KUKA KRL program: HmiToolCheck.src

&ACCESS RVP
&REL 18
&PARAM EDITMASK = *
&PARAM TEMPLATE = C:\KRC\Roboter\Template\vorgabe
DEF HmiToolCheck( )
;FOLD INI;%{PE}
  ;FOLD BASISTECH INI
    GLOBAL INTERRUPT DECL 3 WHEN $STOPMESS==TRUE DO IR_STOPM ( )
    INTERRUPT ON 3
    BAS (#INITMOV,0 )
  ;ENDFOLD (BASISTECH INI)
  ;FOLD USER INI
    ;Make your modifications here

  ;ENDFOLD (USER INI)
;ENDFOLD (INI)

;************************************************
;              CNC Robotics Ltd
;              www.cncrobotics.co.uk
;************************************************
;     Contact: helpdesk@cncrobotics.co.uk
;     Date: 25/09/23
;     Version: 0.12.46
;************************************************
; Description: Program to check if spindle holds
; a tool and drops it if necessary
;************************************************

;If no tool is held then exit program

IF (nToolHeld == 0) THEN
   RETURN
ENDIF

ToolrackMove(nToolHeld) ;Call tool changer to position for drop
ToolRackOpen()		 ;Close tool rack
ToolDrop() 			 ;Run tool drop program
RackSafe()
ToolRackClose()		 ;Close tool rack
HomeRobot()

END
